    |   movel(p[0.514091, -0.111716, -0.000100, 0.000000, -3.141593, 0.000000],accel_mss,speed_ms,0,0.000)
    |   movel(p[0.514271, -0.111866, -0.000100, 0.000000, -3.141593, 0.000000],accel_mss,speed_ms,0,0.000)
    |   movel(p[0.514427, -0.112259, -0.000100, 0.000000, -3.141593, 0.000000],accel_mss,speed_ms,0,0.000)
    |   movel(p[0.514594, -0.113173, -0.000100, 0.000000, -3.141593, 0.000000],accel_mss,speed_ms,0,0.000)
    |   movel(p[0.514523, -0.113998, -0.000100, 0.000000, -3.141593, 0.000000],accel_mss,speed_ms,0,0.000)
    |   movel(p[0.514200, -0.114782, -0.000100, 0.000000, -3.141593, 0.000000],accel_mss,speed_ms,0,0.000)
    |   movel(p[0.513613, -0.115573, -0.000100, 0.000000, -3.141593, 0.000000],accel_mss,speed_ms,0,0.000)
    |   movel(p[0.512987, -0.116165, -0.000100, 0.000000, -3.141593, 0.000000],accel_mss,speed_ms,0,0.000)
    |   movel(p[0.512359, -0.116554, -0.000100, 0.000000, -3.141593, 0.000000],accel_mss,speed_ms,0,0.000)
    |   movel(p[0.511668, -0.116771, -0.000100, 0.000000, -3.141593, 0.000000],accel_mss,speed_ms,0,0.000)
    |   movel(p[0.510851, -0.116843, -0.000100, 0.000000, -3.141593, 0.000000],accel_mss,speed_ms,0,0.000)
    |   movel(p[0.510350, -0.116824, -0.000100, 0.000000, -3.141593, 0.000000],accel_mss,speed_ms,0,0.000)
    |   movel(p[0.509945, -0.116767, -0.000100, 0.000000, -3.141593, 0.000000],accel_mss,speed_ms,0,0.000)
    |   movel(p[0.509583, -0.116661, -0.000100, 0.000000, -3.141593, 0.000000],accel_mss,speed_ms,0,0.000)
    |   movel(p[0.509217, -0.116497, -0.000100, 0.000000, -3.141593, 0.000000],accel_mss,speed_ms,0,0.000)
    |   movel(p[0.508473, -0.116018, -0.000100, 0.000000, -3.141593, 0.000000],accel_mss,speed_ms,0,0.000)
    |   movel(p[0.507748, -0.115372, -0.000100, 0.000000, -3.141593, 0.000000],accel_mss,speed_ms,0,0.000)
    |   movel(p[0.507116, -0.114636, -0.000100, 0.000000, -3.141593, 0.000000],accel_mss,speed_ms,0,0.000)
    |   movel(p[0.506653, -0.113887, -0.000100, 0.000000, -3.141593, 0.000000],accel_mss,speed_ms,0,0.000)
    |   movel(p[0.506318, -0.113033, -0.000100, 0.000000, -3.141593, 0.000000],accel_mss,speed_ms,0,0.000)
    |   speed_ms    = 0.050
    |   movel(p[0.506318, -0.113033, 0.003000, 0.000000, -3.141593, 0.000000],accel_mss,speed_ms,0,blend_radius_m)
    |   speed_ms    = 1.000
    |   movel(p[0.506318, -0.113033, 0.015000, 0.000000, -3.141593, 0.000000],accel_mss,speed_ms,0,blend_radius_m)
    | 
    |   movel(p[0.514600, -0.147080, 0.015000, 0.000000, -3.141593, 0.000000],accel_mss,speed_ms,0,blend_radius_m)
    |   movel(p[0.514600, -0.147080, 0.115000, 0.000000, -3.141593, 0.000000],accel_mss,speed_ms,0,blend_radius_m)
  Halt
